// TIA Portal V20 export
// export: Created 2025-12-01T14:57:42.9011121Z, ExportSetting None, DisplayName Totally Integrated Automation Portal, DisplayVersion V20 Update 3, DisplayName TIA Portal Openness, DisplayVersion V20 Update 3, DisplayName TIA Portal Version Control Interface, DisplayVersion V20 Update 3, DisplayName STEP 7 Professional, DisplayVersion V20 Update 3, DisplayName STEP 7 Safety, DisplayVersion V20 Update 2, DisplayName WinCC Basic/Comfort/Advanced, DisplayVersion V20 Update 3, DisplayName WinCC Professional, DisplayVersion V20 Update 3, DisplayName WinCC Unified, DisplayVersion V20 Update 3
FUNCTION "FC953_Diagnostico_ASi" : Void   // FC953, SCL
{ S7_Optimized_Access := 'TRUE' }
// stored: AutoNumber false, SetENOAutomatically false
   VAR_OUTPUT
      Error_ASI : Bool;
   END_VAR
   VAR_IN_OUT
      Array_ASI3_C1 : Array[*] of "ASI3_Diag_GW";
      Array_ASI3_C2 : Array[*] of "ASI3_Diag_GW";
      Array_ASI5_Flags : Array[*] of "ASI5_Flags";
   END_VAR
   VAR_TEMP
      VarASI : Struct
         InicioArray : UInt;
         FinalArray : UInt;
         Indice : UInt;
      END_STRUCT;
   END_VAR
BEGIN
   //FUNCION QUE BUSCA SI UNA GATEWAY ASI ESTÁ EN ERROR, ACTIVA UN BIT PARA MOSTRAR EN HMI
   REGION Inicializar
       #VarASI.InicioArray := DINT_TO_UINT(LOWER_BOUND(ARR := #Array_ASI3_C2, DIM := 1));
       #VarASI.FinalArray := DINT_TO_UINT(UPPER_BOUND(ARR := #Array_ASI3_C2, DIM := 1));
       #Error_ASI := FALSE;

   END_REGION

   //Busqueda error en ASI-Gatewayes
   FOR #VarASI.Indice := #VarASI.InicioArray TO #VarASI.FinalArray DO
       IF (#Array_ASI3_C1[#VarASI.Indice]."Flags Fault Det" <> 0) OR (#Array_ASI3_C2[#VarASI.Indice]."Flags Fault Det" <> 0) OR
           (#Array_ASI5_Flags[#VarASI.Indice]."C1_FlagsFault" <> 0) OR (#Array_ASI5_Flags[#VarASI.Indice]."C2_FlagsFault" <> 0 <> 0) THEN
           #Error_ASI := TRUE;
           RETURN;
       END_IF;
   END_FOR;
END_FUNCTION
